FUNCTION_BLOCK FB_ABL_115_Pnp
(****************************************************************************************)
(*	TITEL				laden kristall- Modul	    										*)
(*	Status				ungetestet                         								*)
(*	Beschrieb:			Ablaufbeschreibung												*)
(*																						*)
(*	Steps:	self-explained using enum													*)
(***********************************Revisionen*******************************************)
(*	see github blames																	*)
(****************************************************************************************)

VAR_INPUT
    xIN_Reset       : BOOL;          // Schrittkette zurücksetzen 
    xIN_Init        : BOOL;          // Initialisieren
    xIN_Quit        : BOOL;          // Fehler quittieren 
    xIN_Start       : BOOL;          // Startbefehl
    xIN_Sperre      : BOOL;          // FB Sperren 
    xIN_NextStep    : BOOL;          // Nächsten Schritt ausführen 
    xIN_AlarmAktiv  : BOOL;          // Anlage hat Alarm
    xIN_DryCycle    : BOOL;          // Fahren ohne Teile
    xIN_RestartCYCL : BOOL;          // Zyklus erneut starten im STEP, END, LEERFAHREN
    enIN_State      : enState;       // Status Anlage
    tIN_Timeout     : TIME := T#10s; // Timout

    pxFG_Freigabe : POINTER TO BOOL; //Freigabe von Station

    // Application specific
    Mover              : REFERENCE TO FB_Mover;
    xIN_PceReadyToPick : BOOL; // the piece(s) is/are ready to picked
END_VAR
VAR_OUTPUT
    (* standart Ausgänge *)
    xOUT_ErrFlag  : BOOL;        // Error Flag 
    xOUT_Busy     : BOOL;        // Baustein befindet sich im Ablauf 
    xOUT_Done     : BOOL;        // Baustein hat den Ablauf beendet 		
    xOUT_Ready    : BOOL;        // Ready to begin, should be the same state as done	
    xOUT_Timeout  : BOOL;        // Timeout FB 
    xOUT_InitDone : BOOL;        // initialisierung fertig
    xOUT_Wait     : BOOL;        // Wartet auf Bedingung
    iOUT_Step     : ST115_Pnp_e; // Aktueller Schritt 
    sOUT_Step     : STRING;      // Aktueller Schritt but in string format
    bOUT_Error    : BYTE;        // Fehlernummer

    iOUT_ProcessCompletion : INT;  //process completion, express in % (0-100)
    xOUT_MoverFree         : BOOL; // The mover is free to move
    xOUT_PickPiece         : BOOL; // Set to true when a piece is picked

END_VAR
VAR
    (* Standard *)
    (* Schritt *)
    iLastStep : ST115_Pnp_e; // Merker letzter Schritt 
    iPreStep  : ST115_Pnp_e; // Schritt zurück nach Alarm 
    iAktStep  : ST115_Pnp_e; // aktueller Schritt

    // Trigger Starten 
    rtSTART : R_TRIG;
    // Timer TimeOut 
    TON_Timeout : TON;

    (* Bausteine *)

    (* Spezial *)
    fb_axis115_01Y : FB_AxisLM_V1_1;
    fb_axis115_02Z : FB_AxisLIN_V1_1;
    fb_axis115_03Z : FB_AxisLIN_V1_1;

    fb_PnpHorAxis  : FB_LinearMotionMan;
    fb_PnpVerAxisL : FB_LinearMotionMan;
    fb_PnpVerAxisR : FB_LinearMotionMan;

    fb_simu_axis115_01Y : FB_Simu_AxisLM_V1_1;
    fb_simu_axis115_02Z : FB_Simu_AxisLIN_V1_1;
    fb_simu_axis115_03Z : FB_Simu_AxisLIN_V1_1;
	
    fb_gripperLeft    : FB_ZylMo2El_V2_1;
    simu_gripperLeft  : FB_Simu_Zyl2Pos;
    fb_gripperRight   : FB_ZylMo2El_V2_1;
    simu_gripperRight : FB_Simu_Zyl2Pos;

END_VAR
VAR CONSTANT
END_VAR

(*******************************************************************)
(* Trigger  *)
(*******************************************************************)
(* Zurücksetzen *)
IF xIN_RESET THEN
    iPreStep  := ST115_Pnp_e.RESET;
    iOUT_Step := ST115_Pnp_e.RESET;
END_IF;

(* Error Quittieren *)
IF (bOUT_Error <> 0) AND xIN_Quit THEN
    xOUT_ErrFlag := FALSE;
    bOUT_Error   := 0;
    iOUT_Step    := iPreStep;
END_IF;

(*******************************************************************)
(* Timer *)
(*******************************************************************)
TON_Timeout(IN := xIN_NextStep AND (iLastStep = iOUT_Step) (*todo FG *) ,
            PT := tIN_Timeout);

(*******************************************************************)
(* Bausteine *)
(*******************************************************************)
fb_PnpHorAxis(config          := _20_AUTO.recipe.linearAxis[LinearAxis_e.ST115_01Y],
              lrIN_CurrPos    := fb_axis115_01Y.rOUT_ActPos,
              lrIN_Delta_mm   := 0.01,
              iIN_CurrentStep := iOUT_Step,
              iIN_moveNumber  := ST115_PnpHorPos_e._max);

fb_axis115_01Y(enIN_State       := enIN_State,
               parIN_Buttons    := ADR(AXIS.btTeachArAxis),
               xIN_DisButtons   := FALSE,
               xIN_Quit         := xIN_Quit,
               xIN_PARAMok      := TRUE, (*TODO*)
               xIN_FREE         := TRUE,
               xIN_FREE_HOME    := TRUE,
               rIN_POSMIN       := ST115_Axis.const115_01Y.POS_MIN,
               rIN_POSMAX       := ST115_Axis.const115_01Y.POS_MAX,
               rIN_VELOMAX      := ST115_Axis.const115_01Y.VELO_MAX,
               rIN_VELOMANU     := ST115_Axis.const115_01Y.VELO_MANU,
               rIN_VELOOPEN     := ST115_Axis.const115_01Y.VELO_MANU / 4,
               rIN_JogInc       := AXIS.rTeachIncAxis,
               xIN_Execute      := fb_PnpHorAxis.xOUT_Execute,
               xIN_Home         := ST115_Pnp_e.Init_HomeHorizontals = iAktStep,
               xIN_Relative     :=,
               rIN_Position     := TO_REAL(fb_PnpHorAxis.OUT_MoveProfile.lrPosition),
               rIN_Velocity     := TO_REAL(fb_PnpHorAxis.OUT_MoveProfile.lrVelocity),
               rIN_Acceleration := TO_REAL(fb_PnpHorAxis.OUT_MoveProfile.lrAccel),
               rIN_Deceleration := TO_REAL(fb_PnpHorAxis.OUT_MoveProfile.lrDecel),
               rIN_Jerk         := TO_REAL(fb_PnpHorAxis.OUT_MoveProfile.lrJerk),
               xIN_Reset        := (ST115_Pnp_e.RESET = iAktStep) OR xIN_Reset,
               axisIN_REF       := ST115_Axis.axis115_01Y.axis);

fb_simu_axis115_01Y(bIN_AxisCntr        := fb_axis115_01Y.bOUT_AxisCntr,
                    udiIN_HomingTime_ms := 2000,
                    rIN_PosActual       := fb_axis115_01Y.rOUT_ActPos,
                    rIN_PosMax          := ST115_Axis.const115_01Y.POS_MAX,
                    rIN_PosMin          := ST115_Axis.const115_01Y.POS_MIN,
                    rIN_PixMax          := 100,
                    rIN_PixMin          := 0,
                    wOUT_AxisState      => fb_axis115_01Y.wAxisState);

fb_PnpVerAxisL(config          := _20_AUTO.recipe.linearAxis[LinearAxis_e.ST115_02Z],
               lrIN_CurrPos    := fb_axis115_02Z.rOUT_ActPos,
               lrIN_Delta_mm   := 0.01,
               iIN_CurrentStep := iOUT_Step,
               iIN_moveNumber  := ST115_PnpVerPos_e._max);

fb_axis115_02Z(enIN_State     := enIN_State,
               parIN_Buttons  := ADR(AXIS.btTeachArAxis),
               xIN_DisButtons := FALSE,
               xIN_Quit       := xIN_Quit,
               axisIN_REF     := ST115_Axis.axis115_02Z.axis,
               xIN_AX5000     := FALSE,
               xIN_ENC_ABS    := TRUE, // TODO set accordingly
               xIN_PARAMok    := TRUE,
               xIN_FREE       := TRUE,
               xIN_FREE_HOME  := TRUE,
               rIN_POSMIN     := ST115_Axis.const115_02Z.POS_MIN,
               rIN_POSMAX     := ST115_Axis.const115_02Z.POS_MAX,
               rIN_VELOMAX    := ST115_Axis.const115_02Z.VELO_MAX,
               rIN_VELOMANU   := ST115_Axis.const115_02Z.VELO_MANU,
               rIN_VELOOPEN   := ST115_Axis.const115_02Z.POS_MAX / 4,
               rIN_JogInc     := AXIS.rTeachIncAxis,
               rIN_JogVelo    :=,
               xIN_HomeExe    :=,
               xIN_HomeCalib  :=,
               xIN_Execute    := (_20_AUTO.recipe.st115.xUseVerLeft OR (iOUT_Step < ST115_Pnp_e.READY)) AND
                                 (fb_PnpVerAxisL.xOUT_Execute),
               xIN_HomeExe      := NOT CONST.USE_SIMULATION AND (ST115_Pnp_e.Init_HomeVerticals = iAktStep),
               xIN_Relative     :=,
               rIN_Position     := TO_REAL(fb_PnpVerAxisL.OUT_MoveProfile.lrPosition),
               rIN_Velocity     := TO_REAL(fb_PnpVerAxisL.OUT_MoveProfile.lrVelocity),
               rIN_Acceleration := TO_REAL(fb_PnpVerAxisL.OUT_MoveProfile.lrAccel),
               rIN_Deceleration := TO_REAL(fb_PnpVerAxisL.OUT_MoveProfile.lrDecel),
               rIN_Jerk         := TO_REAL(fb_PnpVerAxisL.OUT_MoveProfile.lrJerk),
               xIN_Reset        := (ST115_Pnp_e.RESET = iAktStep) OR xIN_Reset,

               // output
               xOUT_ErrFlag =>,
               xOUT_READY   =>,
               xOUT_DONE    =>,
               bOUT_Error   =>,
               rOUT_ActPos  =>);

fb_simu_axis115_02Z(rIN_PosActual := fb_axis115_02Z.rOUT_ActPos,
                    rIN_PosMax    := ST115_Axis.const115_02Z.POS_MAX,
                    rIN_PosMin    := ST115_Axis.const115_02Z.POS_MIN,
                    rIN_PixMax    := 80,
                    rIN_PixMin    := 0);

fb_PnpVerAxisR(config          := _20_AUTO.recipe.linearAxis[LinearAxis_e.ST115_03Z],
               lrIN_CurrPos    := fb_axis115_03Z.rOUT_ActPos,
               lrIN_Delta_mm   := 0.01,
               iIN_CurrentStep := iOUT_Step,
               iIN_moveNumber  := ST115_PnpVerPos_e._max);

fb_axis115_03Z(enIN_State     := enIN_State,
               parIN_Buttons  := ADR(AXIS.btTeachArAxis),
               xIN_DisButtons := FALSE,
               xIN_Quit       := xIN_Quit,
               xIN_PARAMok    := TRUE, (*TODO*)
               xIN_FREE       := TRUE,
               xIN_FREE_HOME  := TRUE,
               rIN_POSMIN     := ST115_Axis.const115_03Z.POS_MIN,
               rIN_POSMAX     := ST115_Axis.const115_03Z.POS_MAX,
               rIN_VELOMAX    := ST115_Axis.const115_03Z.VELO_MAX,
               rIN_VELOMANU   := ST115_Axis.const115_03Z.VELO_MANU,
               rIN_VELOOPEN   := ST115_Axis.const115_03Z.VELO_MANU / 4,
               rIN_JogInc     := AXIS.rTeachIncAxis,
               xIN_Execute    := (_20_AUTO.recipe.st115.xUseVerRight OR (iOUT_Step < ST115_Pnp_e.READY)) AND
                                 (fb_PnpVerAxisR.xOUT_Execute),
               xIN_HomeExe      := NOT CONST.USE_SIMULATION AND (ST115_Pnp_e.Init_HomeVerticals = iAktStep),
               xIN_Relative     :=,
               rIN_Position     := TO_REAL(fb_PnpVerAxisR.OUT_MoveProfile.lrPosition),
               rIN_Velocity     := TO_REAL(fb_PnpVerAxisR.OUT_MoveProfile.lrVelocity),
               rIN_Acceleration := TO_REAL(fb_PnpVerAxisR.OUT_MoveProfile.lrAccel),
               rIN_Deceleration := TO_REAL(fb_PnpVerAxisR.OUT_MoveProfile.lrDecel),
               rIN_Jerk         := TO_REAL(fb_PnpVerAxisR.OUT_MoveProfile.lrJerk),
               xIN_Reset        := (ST115_Pnp_e.RESET = iAktStep) OR xIN_Reset,
               axisIN_REF       := ST115_Axis.axis115_03Z.axis,
               xIN_AX5000       := FALSE,
               xIN_ENC_ABS      := TRUE); // TODO set accordingly

fb_simu_axis115_03Z(rIN_PosActual := fb_axis115_03Z.rOUT_ActPos,
                    rIN_PosMax    := ST115_Axis.const115_03Z.POS_MAX,
                    rIN_PosMin    := ST115_Axis.const115_03Z.POS_MIN,
                    rIN_PixMax    := 80,
                    rIN_PixMin    := 0);

fb_gripperLeft(xIN_Reset    := xIN_Reset OR (ST115_Pnp_e.RESET = iOUT_Step),
               xIN_Quit     := xIN_Quit,
               xIN_Manu     := enState.StateMANU = enIN_State,
               pbtIN_Button := ADR(HMI.btArManu115[1]),
               xIN_GS       := NOT fb_gripperLeft.xIN_AS,
               xIN_AS       := simu_gripperLeft.xOUT_inAS,
               xIN_FREE     := TRUE,
               xINtoGS      := ST115_Pnp_e.Gripper_open = iOUT_Step,
               xINtoAS      := _20_AUTO.recipe.st115.xUseVerLeft AND (ST115_Pnp_e.Gripper_close = iOUT_Step),
               tIN_ErrAS    := DINT_TO_TIME(_20_AUTO.recipe.cylinder2Pos[StationList_e.ST115]
                                                [ST115_Cylinders_e.GreiferLinks].toAS_alarm_time),
               tIN_ErrGS := DINT_TO_TIME(_20_AUTO.recipe.cylinder2Pos[StationList_e.ST115]
                                             [ST115_Cylinders_e.GreiferLinks].toGS_alarm_time),
               tIN_WaitAS := DINT_TO_TIME(_20_AUTO.recipe.cylinder2Pos[StationList_e.ST115]
                                              [ST115_Cylinders_e.GreiferLinks].toAS_wait_time),
               tIN_WaitGS := DINT_TO_TIME(_20_AUTO.recipe.cylinder2Pos[StationList_e.ST115]
                                              [ST115_Cylinders_e.GreiferLinks].toGS_wait_time));

simu_gripperLeft(xIN_Enable := CONST.USE_SIMULATION,
                 xIN_toGS   := NOT simu_gripperLeft.xIN_toAS,
                 xIN_toAS   := fb_gripperRight.xOUT_VALVE,
                 tIN_GS_ms  := 200,  //ms
                 tIN_AS_ms  := 200); //ms

fb_gripperRight(xIN_Reset    := xIN_Reset OR (ST115_Pnp_e.RESET = iOUT_Step),
                xIN_Quit     := xIN_Quit,
                xIN_Manu     := enState.StateMANU = enIN_State,
                pbtIN_Button := ADR(HMI.btArManu115[2]),
                xIN_GS       := NOT fb_gripperRight.xIN_AS,
                xIN_AS       := simu_gripperRight.xOUT_inAS,
                xIN_FREE     := TRUE,
                xINtoGS      := ST115_Pnp_e.Gripper_open = iOUT_Step,
                xINtoAS      := _20_AUTO.recipe.st115.xUseVerRight AND (ST115_Pnp_e.Gripper_close = iOUT_Step),
                tIN_ErrAS    := DINT_TO_TIME(_20_AUTO.recipe.cylinder2Pos[StationList_e.ST115]
                                                 [ST115_Cylinders_e.GreiferRechts].toAS_alarm_time),
                tIN_ErrGS := DINT_TO_TIME(_20_AUTO.recipe.cylinder2Pos[StationList_e.ST115]
                                              [ST115_Cylinders_e.GreiferRechts].toGS_alarm_time),
                tIN_WaitAS := DINT_TO_TIME(_20_AUTO.recipe.cylinder2Pos[StationList_e.ST115]
                                               [ST115_Cylinders_e.GreiferRechts].toAS_wait_time),
                tIN_WaitGS := DINT_TO_TIME(_20_AUTO.recipe.cylinder2Pos[StationList_e.ST115]
                                               [ST115_Cylinders_e.GreiferRechts].toGS_wait_time));

simu_gripperRight(xIN_Enable := CONST.USE_SIMULATION,
                  xIN_toGS   := NOT simu_gripperRight.xIN_toAS,
                  xIN_toAS   := fb_gripperRight.xOUT_VALVE,
                  tIN_GS_ms  := 200,  //ms
                  tIN_AS_ms  := 200); //ms

(*******************************************************************)
(* OUTPUTS *)
(*******************************************************************)
// Error Flag 
xOUT_ErrFlag := (bOUT_Error <> 0);
// Baustein befindet sich im Ablauf 
xOUT_Busy := (iOUT_Step > ST115_Pnp_e.READY) AND (iOUT_Step < ST115_Pnp_e.DONE);
// Baustein hat den Ablauf beendet
xOUT_Done := (iOUT_Step = ST115_Pnp_e.DONE);
// Process ready
xOUT_Ready := (iOUT_Step = ST115_Pnp_e.READY);
// Timeout FB 				 		
xOUT_Timeout := TON_Timeout.Q;
// Itialisierung fertig			
xOUT_InitDone := (iOUT_Step = ST115_Pnp_e.READY);
// Aktueller Schritt			
iOUT_Step := iOUT_Step; //Im Ablauf gesetzt		
sOUT_Step := TO_STRING(iOUT_Step);
//Fehlernummer	 
bOUT_Error := bOUT_Error; //Im Ablauf/FB gesetzt	
(* Warte (alle Schritte wo auf FG oder Teile gewartet wird) *)
xOUT_Wait := (iOUT_Step = ST115_Pnp_e.DONE);

xOUT_MoverFree := iOUT_Step >= ST115_Pnp_e.MOVER_FREE_OP AND iOUT_Step < ST115_Pnp_e.MOVER_NEEDED_OP;

iOUT_ProcessCompletion := F_GetPercent_2(iAktStep,
                                         ST115_Pnp_e.PnP_Hor_ToRotTablePos,
                                         ST115_Pnp_e.PnP_Hor_ToTrackPos,
                                         ST115_Pnp_e.PnP_Ver_ShuttleDown,
                                         ST115_Pnp_e.PnP_Ver_ShuttleUp);

xOUT_PickPiece := iOUT_Step = ST115_Pnp_e.PnP_Hor_ToTrackPos;

(*******************************************************************)
(* Ablauf *)
(*******************************************************************)

(* Sperren *)
IF xIN_Sperre THEN
    iPreStep  := ST115_Pnp_e.RESET;
    iOUT_Step := ST115_Pnp_e.RESET;
    RETURN;
END_IF;

(* Schritt Merker *)
IF iAktStep <> iOUT_Step THEN
    iLastStep := iAktStep;
    iAktStep  := iOUT_Step;
END_IF

(* START *)
rtSTART(CLK := xIN_Start);

(*******************************************************************)
(* Schrittkette  *)
(*******************************************************************)
CASE iOUT_Step OF

(***** RESET *****)
ST115_Pnp_e.RESET: (* Schritt 0-99 *)
    //Initialisierungen
    //Start Init Ablauf
    IF xIN_Init THEN
        iOUT_Step := ST115_Pnp_e.INIT;
        //Start Manu Ablauf
    ELSIF enIN_State = StateMANU AND xIN_NextStep THEN
        iOUT_Step := ST115_Pnp_e.INIT;
    END_IF;

(***** INIT *****)
ST115_Pnp_e.INIT: (* Grundstellung ? *)
    IF CONST.USE_SIMULATION THEN
        iOUT_Step := ST115_Pnp_e.Init_VerticalsUp;
    ELSE
        iOUT_Step := ST115_Pnp_e.Init_HomeVerticals;
    END_IF;

ST115_Pnp_e.Init_HomeVerticals:
    fb_axis115_02Z.rIN_Velocity := _20_AUTO.recipe.linearAxis[LinearAxis_e.ST115_02Z].movesList[0].lrVelocity;
    fb_axis115_03Z.rIN_Velocity := _20_AUTO.recipe.linearAxis[LinearAxis_e.ST115_03Z].movesList[0].lrVelocity;

    IF fb_axis115_02Z.xOUT_DONE AND fb_axis115_03Z.xOUT_DONE THEN
        iOUT_Step := ST115_Pnp_e.Init_VerticalsUp;
    END_IF

ST115_Pnp_e.Init_VerticalsUp:
    IF fb_PnpVerAxisL.MoveTo(ST115_PnpVerPos_e.UpEmpty).xOUT_InPos AND
       fb_PnpVerAxisR.MoveTo(ST115_PnpVerPos_e.UpEmpty).xOUT_InPos THEN
        IF fb_axis115_01Y.xOUT_READY OR fb_axis115_01Y.xOUT_HOMED THEN
            iOUT_Step := ST115_Pnp_e.Init_HorizontalsToTrack;
        ELSE
            iOUT_Step := ST115_Pnp_e.Init_HomeHorizontals;
        END_IF
    END_IF

ST115_Pnp_e.Init_HomeHorizontals:
    fb_axis115_01Y.rIN_Velocity := _20_AUTO.recipe.linearAxis[LinearAxis_e.ST115_01Y].movesList[0].lrVelocity;

    IF fb_axis115_01Y.xOUT_HOMED THEN
        iOUT_Step := ST115_Pnp_e.Init_HorizontalsToTrack;
    END_IF

ST115_Pnp_e.Init_HorizontalsToTrack:
    IF fb_PnpHorAxis.MoveTo(ST115_PnpHorPos_e.GS).xOUT_InPos THEN
        iOUT_Step := ST115_Pnp_e.READY;
    END_IF

(***** READY / INIT DONE *****)
ST115_Pnp_e.READY:    (* Start AUTO,END,LEER,STEP *)
    IF xIN_Start THEN //IF rtSTART.Q THEN
        iOUT_Step := ST115_Pnp_e.START;
    END_IF

(***** START  ZYKLISCH *****)
ST115_Pnp_e.START: (*  *)
    IF xIN_NextStep AND pxFG_Freigabe^ THEN
        iOUT_Step := ST115_Pnp_e.PnP_Hor_ToRotTablePos;
    END_IF;

ST115_Pnp_e.PnP_Hor_ToRotTablePos:
    IF xIN_NextStep AND fb_PnpHorAxis.MoveTo(ST115_PnpHorPos_e.AS).xOUT_InPos THEN
        iOUT_Step := ST115_Pnp_e.PnP_WaitOnFeeder;
    END_IF

ST115_Pnp_e.PnP_WaitOnFeeder:
    IF xIN_PceReadyToPick THEN
        iOUT_Step := ST115_Pnp_e.PnP_Ver_RotTableDown;
    END_IF

ST115_Pnp_e.PnP_Ver_RotTableDown:
    IF xIN_NextStep AND
       (fb_PnpVerAxisL.MoveTo(ST115_PnpVerPos_e.DownEmpty).xOUT_InPos OR
       NOT _20_AUTO.recipe.st115.xUseVerLeft) AND
       (fb_PnpVerAxisR.MoveTo(ST115_PnpVerPos_e.DownEmpty).xOUT_InPos OR
       NOT _20_AUTO.recipe.st115.xUseVerRight) THEN
        iOUT_Step := ST115_Pnp_e.Gripper_close;
    END_IF;

ST115_Pnp_e.Gripper_close:
    IF xIN_NextStep AND
       (NOT _20_AUTO.recipe.st115.xUseVerLeft OR fb_gripperLeft.xOUT_inAS) AND
       (NOT _20_AUTO.recipe.st115.xUseVerRight OR fb_gripperRight.xOUT_inAS) THEN
        iOUT_Step := ST115_Pnp_e.PnP_Ver_RotTableUp;
    END_IF;

ST115_Pnp_e.PnP_Ver_RotTableUp:
    IF xIN_NextStep AND
       (fb_PnpVerAxisL.MoveTo(ST115_PnpVerPos_e.UpFull).xOUT_InPos OR
       NOT _20_AUTO.recipe.st115.xUseVerLeft) AND
       (
       fb_PnpVerAxisR.MoveTo(ST115_PnpVerPos_e.UpFull).xOUT_InPos OR
       NOT _20_AUTO.recipe.st115.xUseVerRight
           ) THEN
        iOUT_Step := ST115_Pnp_e.PnP_Hor_ToTrackPos;
    END_IF;

ST115_Pnp_e.PnP_Hor_ToTrackPos:
    IF xIN_NextStep AND fb_PnpHorAxis.MoveTo(ST115_PnpHorPos_e.GS).xOUT_InPos THEN
        iOUT_Step := ST115_Pnp_e.waitOnMover;
    END_IF

ST115_Pnp_e.waitOnMover: (*  *)
    IF xIN_NextStep AND __ISVALIDREF(Mover) THEN
        iOUT_Step := ST115_Pnp_e.PnP_Ver_ShuttleDown;
    END_IF;

ST115_Pnp_e.PnP_Ver_ShuttleDown:
    IF xIN_NextStep AND
       (fb_PnpVerAxisL.MoveTo(ST115_PnpVerPos_e.DownFullQuick).xOUT_InPos OR
       NOT _20_AUTO.recipe.st115.xUseVerLeft) AND
       (fb_PnpVerAxisR.MoveTo(ST115_PnpVerPos_e.DownFullQuick).xOUT_InPos OR
       NOT _20_AUTO.recipe.st115.xUseVerRight) THEN
        iOUT_Step := ST115_Pnp_e.PnP_Ver_ShuttleTorqueControl;
    END_IF;

// We need a fb that enables for us torque control. Here we just go a bit further
ST115_Pnp_e.PnP_Ver_ShuttleTorqueControl:
    IF xIN_NextStep AND
       (fb_PnpVerAxisL.MoveTo(ST115_PnpVerPos_e.DownFullTorqueControl).xOUT_InPos OR
       NOT _20_AUTO.recipe.st115.xUseVerLeft) AND
       (fb_PnpVerAxisR.MoveTo(ST115_PnpVerPos_e.DownFullTorqueControl).xOUT_InPos OR
       NOT _20_AUTO.recipe.st115.xUseVerRight) THEN
        iOUT_Step := ST115_Pnp_e.Gripper_open;
    END_IF;

ST115_Pnp_e.Gripper_open:
    IF xIN_NextStep AND fb_gripperLeft.xOUT_inGS AND fb_gripperRight.xOUT_inGS THEN
        iOUT_Step := ST115_Pnp_e.PnP_Ver_ShuttleUp;
    END_IF;

ST115_Pnp_e.PnP_Ver_ShuttleUp:
    IF xIN_NextStep AND
       (fb_PnpVerAxisL.MoveTo(ST115_PnpVerPos_e.UpEmpty).xOUT_InPos OR
       NOT _20_AUTO.recipe.st115.xUseVerLeft) AND
       (fb_PnpVerAxisR.MoveTo(ST115_PnpVerPos_e.UpEmpty).xOUT_InPos OR
       NOT _20_AUTO.recipe.st115.xUseVerRight) THEN
        iOUT_Step := ST115_Pnp_e.SYNC_MOVER_LEAVE;
    END_IF;

ST115_Pnp_e.SYNC_MOVER_LEAVE:
    // The mover needs to be taken by MoverMan
    IF NOT __ISVALIDREF(Mover) THEN
        iOUT_Step := ST115_Pnp_e.DONE;
    END_IF

(***** DONE *****)
ST115_Pnp_e.DONE: (* Letzter Schritt  *)
    IF NOT xIN_AlarmAktiv THEN
        //AUTO
        IF (enIN_State = StateAUTO) AND xIN_RestartCYCL THEN
            iOUT_Step := ST115_Pnp_e.START;
            //STEP / END / LEERFAHREN restart
        ELSIF (enIN_State < StateAUTO) AND (enIN_State >= enState.StateSTEP) AND xIN_RestartCYCL THEN
            iOUT_Step := ST115_Pnp_e.START;
            //STEP / END / LEERFAHREN fertig
        ELSIF (enIN_State = StateREADY) THEN
            iOUT_Step := ST115_Pnp_e.READY;
        END_IF;
    END_IF;

(************ ERROR *************)
ST115_Pnp_e.ERROR: (* ERROR *) ;

END_CASE;

END_FUNCTION_BLOCK

(* stored: Version 1.1.0.1, ProductVersion 3.1.4024.6
   POU FB_ABL_115_Pnp: Id {23721403-6c63-46e6-9cd6-6373b9d6d255}, SpecialFunc None *)
